FUNCTION_BLOCK EQ_Pump (* Filling pump; none is wired yet, so it has no outputs and dispensing is a time at the station's flow rate; equipment IO: owns its IO points, writes the output values its holder sends, reads its inputs every cycle and reports changes *)
  (* Standard: 61499-2 *)
  (* Version 0.1, 2026-09-28, Project contributors, AAU Smart Production Lab *)
  PACKAGE filling;
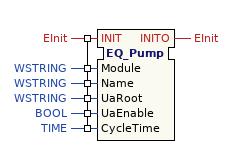
  EVENT_INPUT
    INIT : EInit WITH Module, Name, UaRoot, UaEnable, CycleTime;
  END_EVENT
  EVENT_OUTPUT
    INITO : EInit;
  END_EVENT
  VAR_INPUT
    Module : WSTRING;
    Name : WSTRING := "Pump";
    UaRoot : WSTRING;
    UaEnable : BOOL;
    CycleTime : TIME := T#50ms;
  END_VAR
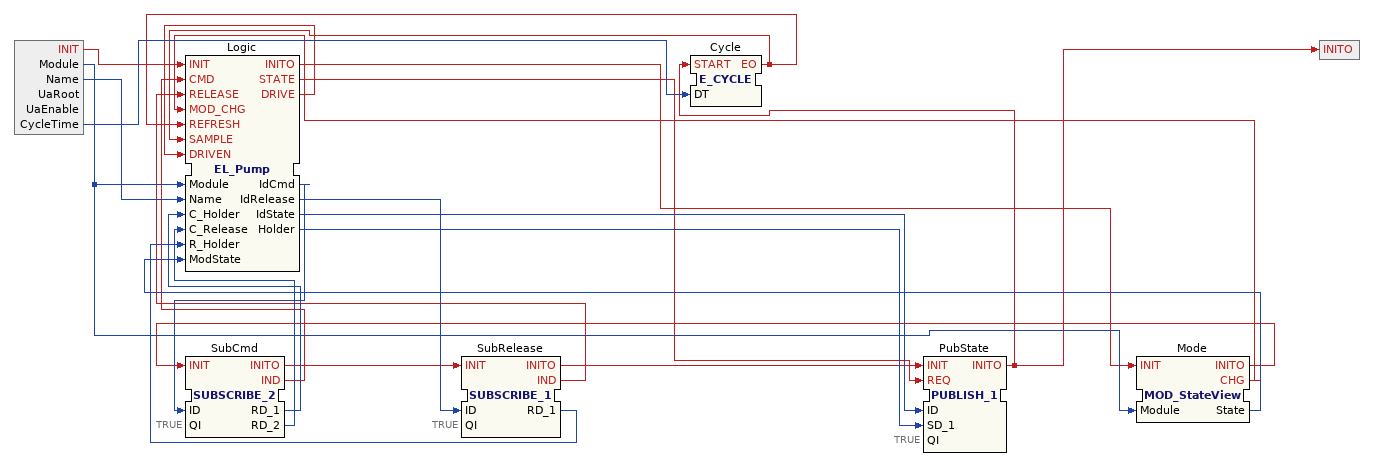
  (* Group Core: One holder at a time, break before make, all off on release or abort; scanned every CycleTime *)
  (* Group Channels: Local channels to and from the skills (cmd, release, state), the module's state, and the inputs over OPC UA *)
  FBS
    Logic : filling::EL_Pump; {SET_ATTRIBUTE(GroupName, Core)}
    Cycle : iec61499::events::E_CYCLE; {SET_ATTRIBUTE(GroupName, Core)}
    Mode : modlib::MOD_StateView; {SET_ATTRIBUTE(GroupName, Channels)}
    SubCmd : iec61499::net::SUBSCRIBE_2(QI := TRUE); {SET_ATTRIBUTE(GroupName, Channels)}
    SubRelease : iec61499::net::SUBSCRIBE_1(QI := TRUE); {SET_ATTRIBUTE(GroupName, Channels)}
    PubState : iec61499::net::PUBLISH_1(QI := TRUE); {SET_ATTRIBUTE(GroupName, Channels)}
  END_FBS
  EVENT_CONNECTIONS
    INIT TO Logic.INIT;
    Logic.INITO TO Mode.INIT;
    Mode.INITO TO SubCmd.INIT;
    SubCmd.INITO TO SubRelease.INIT;
    SubRelease.INITO TO PubState.INIT;
    PubState.INITO TO Cycle.START;
    PubState.INITO TO INITO;
    SubCmd.IND TO Logic.CMD;
    SubRelease.IND TO Logic.RELEASE;
    Mode.CHG TO Logic.MOD_CHG;
    Cycle.EO TO Logic.REFRESH;
    Cycle.EO TO Logic.SAMPLE;
    Logic.STATE TO PubState.REQ;
    Logic.DRIVE TO Logic.DRIVEN;
  END_CONNECTIONS
  DATA_CONNECTIONS
    Module TO Logic.Module;
    Name TO Logic.Name;
    Module TO Mode.Module;
    Logic.IdCmd TO SubCmd.ID;
    Logic.IdRelease TO SubRelease.ID;
    Logic.IdState TO PubState.ID;
    CycleTime TO Cycle.DT;
    SubCmd.RD_1 TO Logic.C_Holder;
    SubCmd.RD_2 TO Logic.C_Release;
    SubRelease.RD_1 TO Logic.R_Holder;
    Mode.State TO Logic.ModState;
    Logic.Holder TO PubState.SD_1;
  END_CONNECTIONS
END_FUNCTION_BLOCK
